// TIA Portal V16 export
// export: Created 2024-09-05T15:58:42.0482152Z, ExportSetting WithDefaults, DisplayName Totally Integrated Automation Portal, DisplayVersion V16 Update 6, DisplayName TIA Portal Version Control Interface, DisplayVersion V16 Update 2, DisplayName TIA Portal Openness, DisplayVersion V16 Update 6, DisplayName STEP 7 Professional, DisplayVersion V16 Update 6, DisplayName STEP 7 Safety, DisplayVersion V16, DisplayName WinCC Advanced, DisplayVersion V16 Update 6
VAR_GLOBAL   // PLC tag table "Hydraulic"
   iOilTemperature50 AT %I10.0 : Bool;   // cooling only - motor running
   iOilTemperature65 AT %I10.1 : Bool;   // motor stop
   iOilHighLevekOK AT %I10.2 : Bool;
   iOilLowLevelOK AT %I10.3 : Bool;   // stop motor if NOK
   iOilFilter1 AT %I10.4 : Bool;
   iOilFilter2 AT %I10.5 : Bool;
   iOilPressureCupping AT %I10.6 : Bool;
   qHydraulicReductionValveCupforming AT %Q10.1 : Bool;
   aiCupformingLeft AT %IW204 : Int;
   aiCupformingRight AT %IW206 : Int;
   qaCupforming1 AT %QW200 : Int;
   qaCupforming2 AT %QW202 : Int;
   qaReductionCupforming AT %QW204 : Int;
   qHydraulicKM20 AT %Q2.0 : Bool;
   qHydraulicKM21 AT %Q2.1 : Bool;
   iHydraulicCircuitBreakerQ2off AT %I2.4 : Bool;
END_VAR
